// TIA Portal project "Paint mixer" (V16)

(* hardware
DEVICE "S7-1200 station_1"  S7-1200 Station
   slot 0: "Rack_0"  S7-1200 Rack  Rack  V1.0
   slot 1: "PLC_1"  CPU 1214C AC/DC/Rly  6ES7 214-1BG40-0XB0  V4.2
DEVICE "PC-System_1"  SIMATIC PC station
   slot 0: "SIMATIC PC station"  Rail  SIMATIC PC-Station  V1.0
      slot 125: "Stationmanager"  Station_Manager  V6.0.4
   slot 2: "IE general_1"  IE General  IE_CP  V8.2.0
   slot 3: "HMI_RT_1"  WinCC RT Advanced  6AV2 104-0xxxx-xxxx  16.0.0.0
      slot 33792: "Computer interface"  Host interface
*)

// ===== PLC "PLC_1"  CPU 1214C AC/DC/Rly =====

ORGANIZATION_BLOCK "Main"   // OB1, LAD, ProgramCycle
TITLE = "Main Program Sweep (Cycle)"
{ S7_Optimized_Access := 'TRUE' }
VERSION : 0.1
   VAR_INPUT
      Initial_Call : Bool;   // Initial call of this OB
      Remanence : Bool;   // =True, if remanent data are available
   END_VAR
BEGIN
END_ORGANIZATION_BLOCK

(* ===== HMI "HMI_RT_1" =====
system functions are stored by id; their names below are inferred from use

Template "Template_1" 1980x1080
   TextField "Text field_1" at 804,7 size 349x59; Text 'HỆ THỐNG PHA MÀU TỰ ĐỘNG'
   Switch "Template_Switch_1" at 39,96 size 122x61; CaptionText 'SIMULATION'; TextOff 'OFF'; TextOn 'ON'
   GraphicView "Template_Graphic view_1" at 112,547 size 187x105; Picture "Graphic_1"
   GraphicView "Template_Graphic view_2" at 667,270 size 77x74; Picture "Graphic_2"
   GraphicView "Template_Graphic view_3" at 325,195 size 101x256; Picture "Graphic_5"
   GraphicView "Template_Graphic view_6" at 763,261 size 67x43; Picture "Graphic_7"
   GraphicView "Template_Graphic view_5" at 787,547 size 389x300; Picture "Graphic_8"
   GraphicView "Template_Graphic view_4" at 925,422 size 116x238; Picture "Graphic_4"
   GraphicView "Template_Graphic view_7" at 513,206 size 148x144; Picture "Graphic_9"
   GraphicView "Template_Graphic view_8" at 1244,261 size 67x43; Picture "Graphic_7"
   GraphicView "Template_Graphic view_9" at 1235,351 size 67x43; Picture "Graphic_7"
   GraphicView "Template_Graphic view_10" at 1236,451 size 67x43; Picture "Graphic_7"
   GraphicView "Template_Graphic view_12" at 1592,81 size 98x112; Picture "Graphic_8"
   GraphicView "Template_Graphic view_13" at 1787,81 size 98x112; Picture "Graphic_8"
   TextField "Template_Text field_1" at 1360,24 size 119x58; Text 'MÀU ĐỎ'
   GraphicView "Template_Graphic view_11" at 1350,83 size 98x112; Picture "Graphic_8"
   Switch "Template_Switch_2" at 176,96 size 124x62; TextOn 'ON'; CaptionText 'SIMULATION'; TextOff 'OFF'
   TextField "Template_Text field_2" at 1592,22 size 119x58; Text 'MÀU VÀNG'
   TextField "Template_Text field_3" at 1787,22 size 119x58; Text 'MÀU XANH'
   TextField "Text field_2" at 82,36 size 206x41; Text 'Bảng điều khiển'
   Bar "Template_Bar_1" at 341,251 size 52x139; MinimumValue 0; MaximumValue 100

screen "Screen_1" 1980x1080
   TextField "Text field_1" at 368,4 size 328x29; Text 'HỆ THỐNG PHA MÀU TỰ ĐỘNG'
   TextField "Text field_2" at 437,39 size 191x18; Text 'PLC S71200 - Tia portal V15.1'
   SymbolLibrary "Symbol library_1" at 36,654 size 229x41
      Appearance <- "Q_BT"
   SymbolLibrary "Symbol library_2" at 206,654 size 229x41
      Appearance <- "Q_BT"
   SymbolLibrary "Symbol library_3" at 371,654 size 229x41
      Appearance <- "Q_BT"
   SymbolLibrary "Symbol library_4" at 541,654 size 229x41
      Appearance <- "Q_BT"
   SymbolLibrary "Symbol library_5" at 713,654 size 229x41
      Appearance <- "Q_BT"
   SymbolLibrary "Symbol library_6" at 883,654 size 229x41
      Appearance <- "Q_BT"
   SymbolLibrary "Symbol library_7" at 1053,654 size 229x41
      Appearance <- "Q_BT"
   SymbolLibrary "Symbol library_8" at 90,693 size 48x60
      Appearance <- "Q_BT"
   SymbolLibrary "Symbol library_9" at 393,153 size 103x148
   SymbolLibrary "Symbol library_12" at 610,332 size 164x167
      Appearance <- "Q_Khuay"
   SymbolLibrary "Symbol library_14" at 658,316 size 72x105
      Appearance <- "Q_Khuay"
   SymbolLibrary "Symbol library_15" at 660,275 size 79x81
      Appearance <- "Q_Khuay"
   SymbolLibrary "Symbol library_13" at 819,33 size 79x89
   Polyline "Polyline_1" at 741,122 size 117x209
      Appearance <- "Q_Van_Nuoc_2"
   SymbolLibrary "Symbol library_17" at 845,176 size 66x58
      Appearance <- "Q_Bom_2"
   SymbolLibrary "Symbol library_16" at 770,179 size 41x47
      Appearance <- "Q_Van_Nuoc_2"
   SymbolLibrary "Symbol library_18" at 1019,33 size 79x89
   Polyline "Polyline_2" at 753,122 size 304x208
      Appearance <- "Q_Van_Nuoc_3"
   SymbolLibrary "Symbol library_21" at 1046,176 size 66x58
      Appearance <- "Q_Bom_3"
   SymbolLibrary "Symbol library_22" at 971,179 size 41x47
      Appearance <- "Q_Van_Nuoc_3"
   SymbolLibrary "Symbol library_19" at 1227,33 size 79x89
   Polyline "Polyline_3" at 762,122 size 503x210
      Appearance <- "Q_Van_Nuoc_4"
   SymbolLibrary "Symbol library_20" at 1254,176 size 66x58
      Appearance <- "Q_Bom_4"
   SymbolLibrary "Symbol library_23" at 1179,179 size 41x47
      Appearance <- "Q_Van_Nuoc_4"
   SymbolLibrary "Symbol library_24" at 868,104 size 37x16
      Appearance <- "M_CB_Low_2"
   SymbolLibrary "Symbol library_25" at 1068,104 size 37x16
      Appearance <- "M_CB_Low_3"
   SymbolLibrary "Symbol library_26" at 1276,104 size 37x16
      Appearance <- "M_CB_Low_4"
   SymbolLibrary "Symbol library_27" at 743,357 size 37x16
      Appearance <- "M_CB_High_5"
   SymbolLibrary "Symbol library_28" at 751,397 size 37x16
      Appearance <- "M_CB_Middle_5"
   SymbolLibrary "Symbol library_29" at 727,453 size 37x16
      Appearance <- "M_CB_Low_5"
   Polyline "Polyline_4" at 494,469 size 182x110
      Appearance <- "Q_Van_Nuoc_5"
   SymbolLibrary "Symbol library_30" at 546,483 size 41x47
      Appearance <- "Q_Van_Nuoc_5"
   Polyline "Polyline_5" at 708,469 size 115x94
      Appearance <- "Q_Van_Nuoc_6"
   SymbolLibrary "Symbol library_31" at 770,483 size 41x47
      Appearance <- "Q_Van_Nuoc_6"
   SymbolLibrary "Symbol library_32" at 1050,473 size 31x82
      Visibility <- "Q_Van_Khi_3"
   SymbolLibrary "Symbol library_33" at 1050,473 size 31x46
   SymbolLibrary "Symbol library_35" at 926,558 size 94x30
      Visibility <- "Q_Van_Khi_2"
   SymbolLibrary "Symbol library_36" at 927,558 size 53x30
   SymbolLibrary "Symbol library_34" at 517,587 size 37x16
      Appearance <- "M_CB2"
   SymbolLibrary "Symbol library_37" at 1094,588 size 37x16
      Appearance <- "M_CB3"
   SymbolLibrary "Symbol library_38" at 1232,588 size 37x16
      Appearance <- "M_CB4"
   Polyline "Polyline_6" at 487,184 size 158x149
      Appearance <- "Q_Van_Nuoc_1"
   SymbolLibrary "Symbol library_39" at 517,199 size 66x58
      Appearance <- "Q_Bom_1"
   SymbolLibrary "Symbol library_10" at 570,148 size 41x47
      Appearance <- "Q_Van_Nuoc_1"
   SymbolLibrary "Symbol library_11" at 460,251 size 37x16
      Appearance <- "M_CB_Low_1"
   TextField "Text field_3" at 492,261 size 26x17; Text 'CB1'
   TextField "Text field_4" at 898,118 size 26x17; Text 'CB2'
   TextField "Text field_5" at 1098,118 size 26x17; Text 'CB3'
   TextField "Text field_6" at 1298,118 size 26x17; Text 'CB4'
   TextField "Text field_10" at 737,30 size 51x17; Text 'MÀU ĐỎ'
   TextField "Text field_13" at 850,236 size 51x17; Text 'BƠM ĐỎ'
   TextField "Text field_14" at 1042,236 size 64x17; Text 'BƠM VÀNG'
   TextField "Text field_15" at 1258,236 size 64x17; Text 'BƠM XANH'
   TextField "Text field_16" at 773,224 size 35x17; Text 'V. ĐỎ'
   TextField "Text field_17" at 973,224 size 48x17; Text 'V. VÀNG'
   TextField "Text field_18" at 1177,224 size 48x17; Text 'V. XANH'
   TextField "Text field_19" at 776,356 size 26x17; Text 'CB7'
   TextField "Text field_20" at 788,396 size 26x17; Text 'CB6'
   TextField "Text field_21" at 764,451 size 26x17; Text 'CB5'
   TextField "Text field_22" at 669,256 size 54x17; Text 'ĐC TRỘN'
   TextField "Text field_23" at 568,129 size 62x17; Text 'VAN NƯỚC'
   TextField "Text field_24" at 528,260 size 66x17; Text 'BƠM NƯỚC'
   TextField "Text field_25" at 413,134 size 62x17; Text 'BỒN NƯỚC'
   TextField "Text field_26" at 541,457 size 41x17; Text 'V. SƠN'
   TextField "Text field_27" at 770,530 size 43x17; Text 'V. RỬA'
   SymbolLibrary "Symbol library_40" at 211,547 size 22x47
      Appearance <- "M_CB1"
   TextField "Text field_28" at 192,526 size 69x17; Text 'CB LON VÀO'
   TextField "Text field_29" at 540,562 size 45x17; Text 'CB RÓT'
   TextField "Text field_30" at 928,594 size 43x17; Text 'XL NẮP'
   TextField "Text field_31" at 1030,451 size 70x17; Text 'XL ĐẬP NẮP'
   TextField "Text field_32" at 1096,569 size 70x17; Text 'CB DẬP NẮP'
   TextField "Text field_33" at 1235,562 size 75x17; Text 'CB KẾT THÚC'
   TextField "Text field_34" at 261,700 size 119x17; Text 'BĂNG TẢI SẢN PHẨM'
   IOField "I/O field_4" at 953,338 size 45x21; FormatPattern 99999
      ProcessValue <- "Act_Time_Tron"
   TextField "Text field_35" at 997,340 size 22x17; Text '[S]'
   TextField "Text field_36" at 858,340 size 38x17; Text 'CHẠY:'
   IOField "I/O field_5" at 953,364 size 45x21; FormatPattern 99999
      ProcessValue <- "Act_Time_Nghi"
   TextField "Text field_37" at 997,366 size 22x17; Text '[S]'
   TextField "Text field_38" at 858,366 size 36x17; Text 'NGHỈ:'
   IOField "I/O field_6" at 953,390 size 45x21; FormatPattern 99999
      ProcessValue <- "Act_Lap_Lai_Tron"
   TextField "Text field_39" at 997,392 size 22x17; Text '[S]'
   TextField "Text field_40" at 858,392 size 84x17; Text 'LẶP LẠI TRỘN;'
   IOField "I/O field_7" at 953,416 size 45x21; FormatPattern 99999
      ProcessValue <- "Act_Lap_Lai_Rua"
   TextField "Text field_41" at 997,418 size 22x17; Text '[S]'
   TextField "Text field_42" at 858,418 size 79x17; Text 'LẶP LẠI RỬA:'
   TextField "Text field_43" at 47,7 size 112x18; Text 'BẢNG ĐIỀU KHIỂN'
   Button "Button_1" at 6,42 size 69x32; TextOff 'CHẠY'
      on Release: ResetBit("M_Start")
      on Press: SetBit("M_Start")
      Appearance <- "Q_Lamp_Running"
   Button "Button_2" at 6,75 size 69x32; TextOff 'DỪNG'
      on Release: ResetBit("M_Stop")
      on Press: SetBit("M_Stop")
      Appearance <- "Q_Lamp_Stop"
   Button "Button_3" at 6,160 size 194x32; TextOff 'CHỌN MÀU TỰ ĐỘNG'
      on Click: function_efd93a16("Pop-up screen_1", 500, 200, -1, -1, 1)
   Circle "Circle_1" at 83,57 size 38x38
      Appearance <- "Q_Lamp_Running"
   TextField "Text field_44" at 89,69 size 26x15; Text 'RUN'
   Circle "Circle_2" at 122,57 size 38x38
      Appearance <- "Q_Lamp_Stop"
   TextField "Text field_45" at 125,69 size 33x15; Text 'STOP'
   Circle "Circle_3" at 162,57 size 38x38
      Appearance <- "Q_Lamp_Fault"
   TextField "Text field_46" at 162,69 size 39x15; Text 'FAULT'
   TextField "Text field_47" at 42,215 size 122x18; Text 'CÀI ĐẶT THÔNG SỐ'
   IOField "I/O field_8" at 122,247 size 45x21; FormatPattern 99999
      ProcessValue <- "Setting_So_Me"
   TextField "Text field_48" at 166,249 size 31x17; Text '[MẺ]'
   TextField "Text field_52" at 7,249 size 57x17; Text 'MẺ TRỘN:'
   IOField "I/O field_9" at 122,271 size 45x21; FormatPattern 999999999.99
      ProcessValue <- "Setting_Tile_Red"
   TextField "Text field_49" at 166,273 size 28x17; Text '[TL]'
   TextField "Text field_50" at 7,273 size 55x17; Text 'TỈ LỆ ĐỎ:'
   IOField "I/O field_10" at 122,295 size 45x21; FormatPattern 999999999.99
      ProcessValue <- "Setting_Tile_Yellow"
   TextField "Text field_51" at 166,297 size 28x17; Text '[TL]'
   TextField "Text field_53" at 7,297 size 70x17; Text 'TỶ LỆ VÀNG:'
   IOField "I/O field_11" at 122,319 size 45x21; FormatPattern 999999999.99
      ProcessValue <- "Setting_Tile_Green"
   TextField "Text field_54" at 166,321 size 28x17; Text '[TL]'
   TextField "Text field_55" at 7,321 size 70x17; Text 'TỶ LỆ XANH:'
   IOField "I/O field_12" at 122,343 size 45x21; FormatPattern 999999999.99
      ProcessValue <- "Setting_Total"
   TextField "Text field_56" at 166,345 size 31x17; Text '[ML]'
   TextField "Text field_57" at 7,345 size 88x17; Text 'TRỌNG LƯỢNG:'
   IOField "I/O field_13" at 122,367 size 45x21; FormatPattern 999999999.99
      ProcessValue <- "Setting_Quy_Doi"
   TextField "Text field_58" at 166,369 size 22x17; Text '[S]'
   TextField "Text field_59" at 7,369 size 82x17; Text 'QUY ĐỔI 1ML:'
   IOField "I/O field_14" at 122,391 size 45x21; FormatPattern 99999
      ProcessValue <- "Setting_Time_Tron"
   TextField "Text field_60" at 166,393 size 22x17; Text '[S]'
   TextField "Text field_61" at 7,393 size 69x17; Text 'TIME TRỘN:'
   IOField "I/O field_15" at 122,415 size 45x21; FormatPattern 99999
      ProcessValue <- "Setting_Time_Nghi"
   TextField "Text field_62" at 166,417 size 22x17; Text '[S]'
   TextField "Text field_63" at 7,417 size 67x17; Text 'TIME NGHỈ:'
   IOField "I/O field_16" at 122,439 size 45x21; FormatPattern 99999
      ProcessValue <- "Setting_Lap_Lai_Tron"
   TextField "Text field_64" at 166,441 size 36x17; Text '[LẦN]'
   TextField "Text field_65" at 7,441 size 81x17; Text 'LẶP LẠI TRỘN'
   IOField "I/O field_17" at 122,463 size 45x21; FormatPattern 99999
      ProcessValue <- "Setting_Lap_Lai_Rua"
   TextField "Text field_66" at 166,465 size 36x17; Text '[LẦN]'
   TextField "Text field_67" at 7,465 size 76x17; Text 'LẶP LẠI RỬA'
   TextField "Text field_68" at 1186,308 size 119x18; Text 'DỮ LIỆU HỆ THỐNG'
   IOField "I/O field_18" at 1265,343 size 45x21; FormatPattern 999999999.9
      ProcessValue <- "Setting_Quy_Doi"
   TextField "Text field_69" at 1309,345 size 22x17; Text '[S]'
   TextField "Text field_70" at 1150,345 size 105x17; Text 'SỐ GIÂY QUY ĐỔI:'
   IOField "I/O field_19" at 1265,367 size 45x21; FormatPattern 999999999.9
      ProcessValue <- "Setting_Quy_Doi_Red"
   TextField "Text field_71" at 1309,369 size 22x17; Text '[S]'
   TextField "Text field_72" at 1150,369 size 54x17; Text 'MÀU ĐỎ:'
   IOField "I/O field_20" at 1265,391 size 45x21; FormatPattern 999999999.9
      ProcessValue <- "Setting_Quy_Doi_Yellow"
   TextField "Text field_73" at 1309,393 size 22x17; Text '[S]'
   TextField "Text field_74" at 1150,393 size 67x17; Text 'MÀU VÀNG:'
   IOField "I/O field_21" at 1265,415 size 45x21; FormatPattern 999999999.9
      ProcessValue <- "Setting_Quy_Doi_Green"
   TextField "Text field_75" at 1309,417 size 22x17; Text '[S]'
   TextField "Text field_76" at 1150,417 size 66x17; Text 'MÀY XANH:'
   IOField "I/O field_22" at 1265,439 size 45x21; FormatPattern 99999
      ProcessValue <- "Act_So_Me"
   TextField "Text field_77" at 1309,441 size 31x17; Text '[MẺ]'
   TextField "Text field_78" at 1150,441 size 71x17; Text 'MẺ THỰC TẾ'
   SymbolLibrary "Symbol library_41" at 205,617 size 32x57
      Visibility <- "M_CB1"
   SymbolLibrary "Symbol library_42" at 41,574 size 94x30
      Visibility <- "Q_Van_Khi_1"
   SymbolLibrary "Symbol library_43" at 42,574 size 53x30
   TextField "Text field_79" at 43,610 size 69x17; Text 'XL ĐẨY LON'
   SymbolLibrary "Symbol library_44" at 477,617 size 32x57
      Visibility <- "M_CB2"
   SymbolLibrary "Symbol library_45" at 1050,617 size 32x57
      Visibility <- "M_CB3"
   Rectangle "Rectangle_9" at 234,35 size 87x33
      Appearance <- "TG_Auto_Step1"
   TextField "Text field_80" at 246,42 size 61x18; Text 'RÓT LIỆU'
   Rectangle "Rectangle_10" at 234,99 size 87x33
      Appearance <- "TG_Auto_Step2"
   TextField "Text field_81" at 243,106 size 69x18; Text 'TRỘN LIỆU'
   Rectangle "Rectangle_11" at 234,162 size 87x33
      Appearance <- "TG_Auto_Step3"
   TextField "Text field_82" at 243,169 size 70x18; Text 'CHIẾT RÓT'
   Rectangle "Rectangle_12" at 234,225 size 87x33
      Appearance <- "TG_Auto_Step4"
   TextField "Text field_83" at 245,232 size 65x18; Text 'BƠM RỬA'
   Rectangle "Rectangle_13" at 234,288 size 87x33
      Appearance <- "TG_Auto_Step5"
   TextField "Text field_84" at 239,295 size 77x18; Text 'KHUẤY RỬA'
   Rectangle "Rectangle_14" at 234,351 size 87x33
      Appearance <- "TG_Auto_Step6"
   TextField "Text field_85" at 251,358 size 53x18; Text 'XẢ RỬA'
   Rectangle "Rectangle_15" at 234,414 size 87x33
      Appearance <- "TG_Tron_Xong"
   TextField "Text field_86" at 246,421 size 63x18; Text 'KẾT THÚC'
   Switch "Switch_1" at 533,278 size 50x37; TextOn 'ON'; CaptionText 'Switch'; TextOff 'OFF'
      on SwitchOff: ResetBit("TG_Btt_Manu_Bom_1")
      on SwitchOn: SetBit("TG_Btt_Manu_Bom_1")
      Visibility <- "TG_Btt_Manu"
      ProcessValue <- "TG_Btt_Manu_Bom_1"
   Switch "Switch_2" at 621,142 size 50x37; TextOn 'ON'; CaptionText 'Switch'; TextOff 'OFF'
      on SwitchOff: ResetBit("TG_Btt_Manu_Van_Nuoc_1")
      on SwitchOn: SetBit("TG_Btt_Manu_Van_Nuoc_1")
      Visibility <- "TG_Btt_Manu"
      ProcessValue <- "TG_Btt_Manu_Van_Nuoc_1"
   Switch "Switch_3" at 717,166 size 50x37; TextOn 'ON'; CaptionText 'Switch'; TextOff 'OFF'
      on SwitchOff: ResetBit("TG_Btt_Manu_Van_Nuoc_2")
      on SwitchOn: SetBit("TG_Btt_Manu_Van_Nuoc_2")
      Visibility <- "TG_Btt_Manu"
      ProcessValue <- "TG_Btt_Manu_Van_Nuoc_2"
   Switch "Switch_4" at 877,150 size 50x37; TextOn 'ON'; CaptionText 'Switch'; TextOff 'OFF'
      on SwitchOff: ResetBit("TG_Btt_Manu_Bom_2")
      on SwitchOn: SetBit("TG_Btt_Manu_Bom_2")
      Visibility <- "TG_Btt_Manu"
      ProcessValue <- "TG_Btt_Manu_Bom_2"
   Switch "Switch_5" at 973,238 size 50x37; TextOn 'ON'; CaptionText 'Switch'; TextOff 'OFF'
      on SwitchOff: ResetBit("TG_Btt_Manu_Van_Nuoc_3")
      on SwitchOn: SetBit("TG_Btt_Manu_Van_Nuoc_3")
      Visibility <- "TG_Btt_Manu"
      ProcessValue <- "TG_Btt_Manu_Van_Nuoc_3"
   Switch "Switch_6" at 1069,150 size 50x37; TextOn 'ON'; CaptionText 'Switch'; TextOff 'OFF'
      on SwitchOff: ResetBit("TG_Btt_Manu_Bom_3")
      on SwitchOn: SetBit("TG_Btt_Manu_Bom_3")
      Visibility <- "TG_Btt_Manu"
      ProcessValue <- "TG_Btt_Manu_Bom_3"
   Switch "Switch_7" at 1178,238 size 50x37; TextOn 'ON'; CaptionText 'Switch'; TextOff 'OFF'
      on SwitchOff: ResetBit("TG_Btt_Manu_Van_Nuoc_4")
      on SwitchOn: SetBit("TG_Btt_Manu_Van_Nuoc_4")
      Visibility <- "TG_Btt_Manu"
      ProcessValue <- "TG_Btt_Manu_Van_Nuoc_4"
   Switch "Switch_8" at 1274,150 size 50x37; TextOn 'ON'; CaptionText 'Switch'; TextOff 'OFF'
      on SwitchOff: ResetBit("TG_Btt_Manu_Bom_4")
      on SwitchOn: SetBit("TG_Btt_Manu_Bom_4")
      Visibility <- "TG_Btt_Manu"
      ProcessValue <- "TG_Btt_Manu_Bom_4"
   Switch "Switch_9" at 669,217 size 50x37; TextOn 'ON'; CaptionText 'Switch'; TextOff 'OFF'
      on SwitchOff: ResetBit("TG_Btt_Manu_Khuay")
      on SwitchOn: SetBit("TG_Btt_Manu_Khuay")
      Visibility <- "TG_Btt_Manu"
      ProcessValue <- "TG_Btt_Manu_Khuay"
   Switch "Switch_10" at 811,462 size 50x37; TextOn 'ON'; CaptionText 'Switch'; TextOff 'OFF'
      on SwitchOff: ResetBit("TG_Btt_Manu_Van_Nuoc_6")
      on SwitchOn: SetBit("TG_Btt_Manu_Van_Nuoc_6")
      Visibility <- "TG_Btt_Manu"
      ProcessValue <- "TG_Btt_Manu_Van_Nuoc_6"
   Switch "Switch_11" at 492,474 size 50x37; TextOn 'ON'; CaptionText 'Switch'; TextOff 'OFF'
      on SwitchOff: ResetBit("TG_Btt_Manu_Van_Nuoc_5")
      on SwitchOn: SetBit("TG_Btt_Manu_Van_Nuoc_5")
      Visibility <- "TG_Btt_Manu"
      ProcessValue <- "TG_Btt_Manu_Van_Nuoc_5"
   Switch "Switch_12" at 1092,474 size 50x37; TextOn 'ON'; CaptionText 'Switch'; TextOff 'OFF'
      on SwitchOff: ResetBit("TG_Btt_Manu_Van_Khi_3")
      on SwitchOn: SetBit("TG_Btt_Manu_Van_Khi_3")
      Visibility <- "TG_Btt_Manu"
      ProcessValue <- "TG_Btt_Manu_Van_Khi_3"
   Switch "Switch_13" at 930,510 size 50x37; TextOn 'ON'; CaptionText 'Switch'; TextOff 'OFF'
      on SwitchOff: ResetBit("TG_Btt_Manu_Van_Khi_2")
      on SwitchOn: SetBit("TG_Btt_Manu_Van_Khi_2")
      Visibility <- "TG_Btt_Manu"
      ProcessValue <- "TG_Btt_Manu_Van_Khi_2"
   Switch "Switch_14" at 44,531 size 50x37; TextOn 'ON'; CaptionText 'Switch'; TextOff 'OFF'
      on SwitchOff: ResetBit("TG_Btt_Manu_Van_Khi_1")
      on SwitchOn: SetBit("TG_Btt_Manu_Van_Khi_1")
      Visibility <- "TG_Btt_Manu"
      ProcessValue <- "TG_Btt_Manu_Van_Khi_1"
   Switch "Switch_15" at 94,110 size 107x44; TextOn 'AUTO'; CaptionText 'CHẾ ĐỘ VH'; TextOff 'MANU'
      on SwitchOff: ResetBit("TG_btt_Mode")
      on SwitchOn: SetBit("TG_btt_Mode")
      ProcessValue <- "TG_btt_Mode"
   Switch "Switch_16" at 7,112 size 84x41; TextOn 'ON'; CaptionText 'SIMULATION'; TextOff 'OFF'
      on SwitchOff: ResetBit("TG_Btt_Simulation")
      on SwitchOn: SetBit("TG_Btt_Simulation")
      ProcessValue <- "TG_Btt_Simulation"
   Circle "Circle_4" at 356,74 size 48x48
      Appearance <- "TG_Dieu_Kien_VH"
   TextField "Text field_87" at 362,90 size 36x17; Text 'ĐKVH'
   IOField "I/O field_23" at 743,52 size 45x21; FormatPattern 999999999.99
      ProcessValue <- "Setting_Quy_Doi_Red"
   TextField "Text field_88" at 787,54 size 22x17; Text '[S]'
   TextField "Text field_89" at 708,54 size 28x17; Text 'SET:'
   IOField "I/O field_24" at 743,76 size 45x21; FormatPattern 999999999.99
      ProcessValue <- "Act_Red"
   TextField "Text field_90" at 787,78 size 22x17; Text '[S]'
   TextField "Text field_91" at 708,78 size 30x17; Text 'ACT:'
   TextField "Text field_7" at 929,30 size 64x17; Text 'MÀU VÀNG'
   IOField "I/O field_1" at 943,52 size 45x21; FormatPattern 999999999.99
      ProcessValue <- "Setting_Quy_Doi_Yellow"
   TextField "Text field_92" at 987,54 size 22x17; Text '[S]'
   TextField "Text field_93" at 908,54 size 28x17; Text 'SET:'
   IOField "I/O field_25" at 943,76 size 45x21; FormatPattern 999999999.99
      ProcessValue <- "Act_Yellow"
   TextField "Text field_94" at 987,78 size 22x17; Text '[S]'
   TextField "Text field_95" at 908,78 size 30x17; Text 'ACT:'
   TextField "Text field_11" at 1137,30 size 64x17; Text 'MÀU XANH'
   IOField "I/O field_26" at 1151,52 size 45x21; FormatPattern 999999999.99
      ProcessValue <- "Setting_Quy_Doi_Green"
   TextField "Text field_96" at 1195,54 size 22x17; Text '[S]'
   TextField "Text field_97" at 1116,54 size 28x17; Text 'SET:'
   IOField "I/O field_27" at 1151,76 size 45x21; FormatPattern 999999999.99
      ProcessValue <- "Act_Green"
   TextField "Text field_98" at 1195,78 size 22x17; Text '[S]'
   TextField "Text field_99" at 1116,78 size 30x17; Text 'ACT:'
   Switch "Switch_17" at 159,716 size 50x37; TextOn 'ON'; CaptionText 'Switch'; TextOff 'OFF'
      on SwitchOff: ResetBit("TG_Btt_Manu_BT")
      on SwitchOn: SetBit("TG_Btt_Manu_BT")
      ProcessValue <- "TG_Btt_Manu_BT"
   Group "Group" at 591,233 size 197x144
   SymbolLibrary "Symbol library_47" at 205,617 size 32x57
      Visibility <- "TG_Chai_VT1_2"
      HorizontalMovement <- "Simu_VT_Chai"
   SymbolLibrary "Symbol library_48" at 477,617 size 32x57
      Visibility <- "TG_Chai_VT2_3"
      HorizontalMovement <- "Simu_VT_Chai"
   Group "Group_2" at 1210,611 size 33x62
   Group "Group_1" at 1050,612 size 33x62
   Rectangle "Rectangle_16" at 591,242 size 197x135
      Visibility <- "TG_Tron_Xong"
   TextField "Text field_104" at 733,348 size 31x17; Text '[MẺ]'
      Visibility <- "TG_Tron_Xong"
   IOField "I/O field_29" at 689,346 size 45x21; FormatPattern 99999
      Visibility <- "TG_Tron_Xong"
      ProcessValue <- "Act_So_Me"
   TextField "Text field_105" at 598,348 size 71x17; Text 'MẺ THỰC TẾ'
      Visibility <- "TG_Tron_Xong"
   TextField "Text field_103" at 598,324 size 66x17; Text 'MÀY XANH:'
      Visibility <- "TG_Tron_Xong"
   IOField "I/O field_28" at 689,322 size 45x21; FormatPattern 999999999.9
      Visibility <- "TG_Tron_Xong"
      ProcessValue <- "Setting_Quy_Doi_Green"
   TextField "Text field_102" at 733,324 size 22x17; Text '[S]'
      Visibility <- "TG_Tron_Xong"
   TextField "Text field_100" at 733,300 size 22x17; Text '[S]'
      Visibility <- "TG_Tron_Xong"
   IOField "I/O field_3" at 689,298 size 45x21; FormatPattern 999999999.9
      Visibility <- "TG_Tron_Xong"
      ProcessValue <- "Setting_Quy_Doi_Yellow"
   TextField "Text field_101" at 598,300 size 67x17; Text 'MÀU VÀNG:'
      Visibility <- "TG_Tron_Xong"
   TextField "Text field_12" at 598,276 size 54x17; Text 'MÀU ĐỎ:'
      Visibility <- "TG_Tron_Xong"
   IOField "I/O field_2" at 689,274 size 45x21; FormatPattern 999999999.9
      Visibility <- "TG_Tron_Xong"
      ProcessValue <- "Setting_Quy_Doi_Red"
   TextField "Text field_9" at 733,276 size 22x17; Text '[S]'
      Visibility <- "TG_Tron_Xong"
   Rectangle "Rectangle_17" at 591,233 size 197x31
      Visibility <- "TG_Tron_Xong"
   Button "Button_4" at 756,236 size 29x24; TextOff 'X'
      on Release: ResetBit("M_Stop")
      on Press: SetBit("M_Stop")
      Visibility <- "TG_Tron_Xong"
   TextField "Text field_8" at 598,237 size 119x20; Text 'TB ĐÃ TRỘN XONG'
      Visibility <- "TG_Tron_Xong"
   SymbolLibrary "Symbol library_50" at 1210,616 size 32x57
      Visibility <- "M_CB4"
   Rectangle "Rectangle_19" at 1210,611 size 33x13
      Visibility <- "M_CB4"
   SymbolLibrary "Symbol library_49" at 1050,617 size 32x57
      Visibility <- "TG_Chai_VT3_4"
      HorizontalMovement <- "Simu_VT_Chai"
   Rectangle "Rectangle_18" at 1050,612 size 33x13
      Visibility <- "TG_Chai_VT3_4"
      HorizontalMovement <- "Simu_VT_Chai"
*)